INTERFACE ITF_Blikkenvullijn

END_INTERFACE

(* stored: Version 1.1.0.1, ProductVersion 3.1.4024.12
   Itf ITF_Blikkenvullijn: Id {b0828150-22c5-45c8-9e2c-aea04fc32620} *)
